Staubli VAL3: test.pgx

program test()
begin
  putln("test call")
end
